{attribute addProperty BoxType "EK1100-0000-0018"}
{attribute addProperty Id "Beckhoff_EKx9xxEK1122Beckhoff_EKx9xxEK1122_199990A54464558"}
{attribute addProperty CRC "338708849"}
{attribute addProperty SizeInBites "4464"}
{attribute addProperty SizeInBytes "558"}
TYPE Beckhoff_EKx9xx_14304971 EXTENDS EK1100_179A0949 :
STRUCT
	{attribute addProperty Name "Beckhoff_EKx9xxEK1122"}
	Beckhoff_EKx9xxEK1122 : Beckhoff_EKx9xxEK1122_199990A5;
END_STRUCT
END_TYPE

(* stored: Version 1.2.0.0, ProductVersion 3.1.4024.9
   DUT Beckhoff_EKx9xx_14304971: Id {6fe84759-cf7b-4352-a33b-5fa2bdac387c} *)
